{attribute 'qualified_only'}
VAR_GLOBAL
	CNV_ID_HMI_Old_1:  DINT;
	CNV_ID_HMI:  DINT;
	CNV_ID_HMI_1:  DINT;
	CNV_ID_HMI_Old:  DInt;
	CNV_In_Out_1:  BOOL;
	CNV_Level_Selected:  UInt;
	CNV_Level_Selected_OLD:  UInt;
	CNV_Motor_Actual_Torque:  Real;
	CNV_Motor_Actual_Torque_1:  REAL;
	CNV_Motor_Current_Actual_HMI:  Real;
	CNV_Motor_Current_Actual_HMI_1:  REAL;
	CNV_Motor_Ready:  Bool;
	CNV_Motor_Ready_1:  BOOL;
	CNV_Motor_Status_HMI:  UInt;
	CNV_Motor_Status_HMI_1:  UINT;
	Cnv_Occupied_HMI:  Bool;
	Cnv_Occupied_HMI_1:  BOOL;
	CNV_System_Selected:  UInt;
	CVTD_CNV2_Selected:  UInt;
	Enable_HMI:  Bool;
	Enable_HMI_1:  Bool;
	Enabled_HMI:  Bool;
	Enabled_HMI_1:  Bool;
	Error_HMI:  Bool;
	Error_HMI_1:  Bool;
	HMI_Light_Guard_Bypass:  Bool;
	Light_Guard_Bypass_1:  Bool;
	Light_Guard_Bypass_2:  Bool;
	Manual_Bwd_HMI:  Bool;
	Manual_Bwd_HMI_1:  Bool;
	Manual_Fwd_HMI:  Bool;
	Manual_Fwd_HMI_1:  Bool;
	Manual_Sfty_Stopper_Down_1:  Bool;
	Manual_Sfty_Stopper_Up_1:  Bool;
	Mode_Change_HMI:  UInt;
	Mode_Change_HMI_1:  UInt;
	Mode_HMI:  UInt;
	Mode_HMI_1:  UInt;
	Motor_Direction_HMI:  UInt;
	Motor_Direction_HMI_1:  UInt;
	Motor_Speed_Actual_HMI:  UInt;
	Motor_Speed_Actual_HMI_1:  UInt;
	Motor_Speed_Requested_HMI:  UInt;
	Motor_Speed_Requested_HMI_1:  UInt;
	Ready_For_Task_HMI:  Bool;
	Ready_For_Task_HMI_1:  Bool;
	Reset_HMI:  Bool;
	Reset_HMI_1:  Bool;
	Running_HMI:  Bool;
	Running_HMI_1:  Bool;
	SM_State_HMI:  UInt;
	SM_State_HMI_1:  UInt;
	Start_Transfer_HMI:  Bool;
	Start_Transfer_HMI_1:  Bool;
	Stop_HMI:  Bool;
	Stopped_HMI:  Bool;
	Stopped_HMI_1:  Bool;
	Transfer_From_ID_HMI:  DInt;
	Transfer_From_ID_HMI_1:  DInt;
	Transfer_To_ID_HMI:  DInt;
	Transfer_To_ID_HMI_1:  DInt;
	UpDown_1:  UInt;
	Warning_HMI:  UInt;
	Warning_HMI_1:  UINT;
END_VAR

(* stored: Version 1.1.0.1
   GVL CNV_HMI: Id {b87a538f-d9b3-47dc-bce7-7440947f5e01} *)
